(* PLC project mspindle, Dassault Systèmes ControlBuild 2024x *)
(* stored: creationDateTime 2023-10-03T11:13:47-01:00 *)

PROGRAM drill.mspindle
  VAR_INPUT
    rotationFunction : BOOL := false;
  END_VAR
  VAR_INPUT
    acknowledgePB : BOOL := false;
  END_VAR
  VAR_INPUT
    autoMode : BOOL := false;
    manualMode : BOOL := false;
  END_VAR
  VAR_OUTPUT
    rotationFault : DINT := 0;
  END_VAR

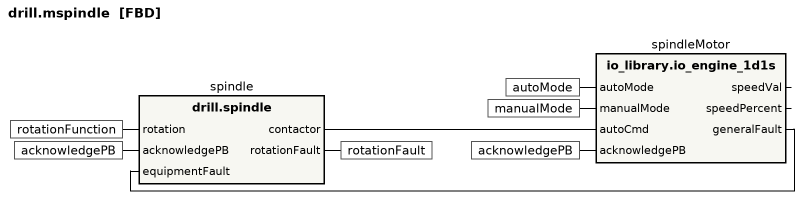
(* FBD diagram, written out as Structured Text *)
spindleMotor(autoMode := autoMode, manualMode := manualMode, autoCmd := spindle.contactor, acknowledgePB := acknowledgePB);
spindle(rotation := rotationFunction, acknowledgePB := acknowledgePB, equipmentFault := spindleMotor.generalFault);
rotationFault := spindle.rotationFault;
END_PROGRAM
